// TIA Portal V18 export
TYPE "UDT_MES_Monitoring"
   STRUCT
      Header : Struct
         Heartbeat_MES : Bool;
         Heartbeat_PLC : Bool;
         MES_Online : Bool;
         MES_HeartbeatTimeout : Bool;
         PLC_HeartbeatTimeout : Bool;
         MES_HeartbeatAge : Time;
         PLC_HeartbeatAge : Time;
      END_STRUCT;
      Station : Array[1..8] of "UDT_MES_Monitoring_station";
      Special : Struct
         StoveCheckInReq : Bool;
         StoveCheckInOk : Bool;
         InProgress : Bool;
         Timeout : Bool;
         Elapsed : Time;
         CountOk : UDInt;
         CountTimeout : UDInt;
      END_STRUCT;
      LastError : Struct
         "Station Number" : Int;
         Code : DInt;
         Text : String[128];
         ActCnt_Errors : Int;
      END_STRUCT;
      Counters : Struct
         TotalDone_CheckIn : UDInt;
         TotalDone_CheckOut : UDInt;
         TotalTimeout_CheckIn : UDInt;
         TotalTimeout_CheckOut : UDInt;
         TotalOK_CheckIn : UDInt;
         TotalNG_CheckIn : UDInt;
         TotalOK_CheckOut : UDInt;
         TotalNG_CheckOut : UDInt;
      END_STRUCT;
   END_STRUCT;
END_TYPE
